// TIA Portal V18 export
// export: Created 2025-12-01T17:51:15.3461758Z, ExportSetting None, DisplayName Totally Integrated Automation Portal, DisplayVersion V18 Update 5, DisplayName TIA Portal Openness, DisplayVersion V18 Update 5, DisplayName TIA Portal Teamcenter Gateway, DisplayVersion V18, DisplayName TIA Portal Version Control Interface, DisplayVersion V18, DisplayName STEP 7 Professional, DisplayVersion V18 Update 5, DisplayName STEP 7 Safety, DisplayVersion V18, DisplayName WinCC Professional, DisplayVersion V18 Update 5
DATA_BLOCK "Robot_DB"   // DB2405
{ S7_Optimized_Access := 'FALSE' }
// stored: AutoNumber false
   VAR
      LoadNG_1 : Array[1..5] of Bool;
      LoadNG_2 : Array[1..5] of Bool;
      LoadNG_3 : Array[1..5] of Bool;
      UnLoadNG_1 : Array[1..5] of Bool;
      UnLoadNG_2 : Array[1..5] of Bool;
      UnLoadNG_3 : Array[1..5] of Bool;
      P : Array[1..16] of Bool;
      RobotFlag_1 : Array[1..8] of Bool;
      RobotFlag_2 : Array[1..8] of Bool;
      RobotFlag_3 : Array[1..8] of Bool;
      RobotSpeed : Array[1..8] of USInt;
      TON : Array[1..18] of TON_TIME;
      Control : Struct
         Robot1GripControl : Bool;
         Robot2GripControl : Bool;
         Robot3GripControl : Bool;
      END_STRUCT;
      Robot_1 : Struct
         PalletCount_1 : Int;
         GripCompareCodeOK_1 : Bool;
         GripCompareCodeOK_2 : Bool;
         GripCompareCodeOK_3 : Bool;
         GripCompareCodeOK_4 : Bool;
         GripCompareCodeOK : Bool;
         Spare_8 : Bool;
         Spare_6 : Bool;
         Spare_7 : Bool;
         SpeedChangeFlag : Bool;
         MasteringTest_Req : Bool;
         BrakeTest_Req : Bool;
         Spare_11 : Bool;
         Spare_12 : Bool;
         Spare_13 : Bool;
         Spare_14 : Bool;
         Spare_15 : Bool;
         SpeedCount : Int;
      END_STRUCT;
      Robot_2 : Struct
         PalletCount_1 : Int;
         PalletCount_2 : Int;
         GripCompareCodeOK_1 : Bool;
         GripCompareCodeOK_2 : Bool;
         GripCompareCodeOK_3 : Bool;
         GripCompareCodeOK_4 : Bool;
         GripCompareCodeOK : Bool;
         Spare_5 : Bool;
         Spare_6 : Bool;
         Spare_7 : Bool;
         SpeedChangeFlag : Bool;
         MasteringTest_Req : Bool;
         BrakeTest_Req : Bool;
         Spare_11 : Bool;
         Spare_12 : Bool;
         Spare_13 : Bool;
         Spare_14 : Bool;
         Spare_15 : Bool;
         SpeedCount : Int;
      END_STRUCT;
      Robot_3 : Struct
         PalletCount_1 : Int;
         PalletCount_2 : Int;
         GripCompareCodeOK_1 : Bool;
         GripCompareCodeOK_2 : Bool;
         GripCompareCodeOK_3 : Bool;
         GripCompareCodeOK_4 : Bool;
         GripCompareCodeOK : Bool;
         Spare_5 : Bool;
         Spare_6 : Bool;
         Spare_7 : Bool;
         SpeedChangeFlag : Bool;
         MasteringTest_Req : Bool;
         BrakeTest_Req : Bool;
         Spare_11 : Bool;
         Spare_12 : Bool;
         Spare_13 : Bool;
         Spare_14 : Bool;
         Spare_15 : Bool;
         SpeedCount : Int;
      END_STRUCT;
   END_VAR
BEGIN
END_DATA_BLOCK
